(* CODESYS project arrayVar_RECOVERED_2024-06-20T13-42-02.project

Project tree, tasks and I/O mapping:
  Device : CODESYS Control Win V3, CODESYS, version 3.5.20.0
    application Application
      libraries: Standard, 3.5.18.0 (System)
      task MainTask (cyclic, interval t#20ms, priority 1) calls PLC_PRG
      function block Flash [LD]
      program PLC_PRG [ST]
*)

// Device/Application/PLC_PRG
PROGRAM PLC_PRG
VAR
	
	// This is an array which keeps the info regarding some sensors
	FArray: ARRAY[0..4] OF Bool := [TRUE, 3(FALSE), TRUE];
	// Real values from sensors
	F2: ARRAY[0..1, 0..1] OF REAL := [11, 0, 6.8, 2.3];
	F3: ARRAY[2..3, 0..1, 1..3, 0..1];
END_VAR

END_PROGRAM

// Device/Application/Flash
FUNCTION_BLOCK Flash
VAR_INPUT
	StartFlsh: BOOL;
	
END_VAR
VAR_OUTPUT
	FlashOut: BOOL;
	
	
END_VAR
VAR
	
	TON_1: TON;
	TON_0: TON;
END_VAR

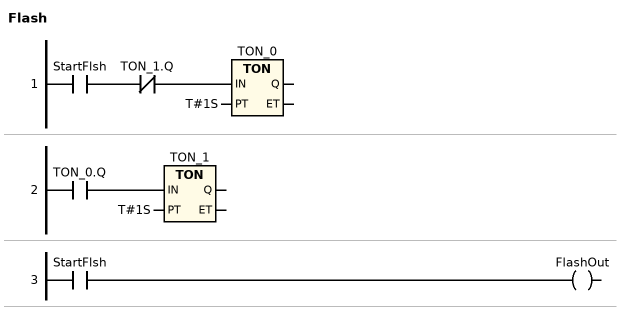
// NETWORK 1
TON_0(IN := StartFlsh AND NOT TON_1.Q, PT := T#1S); // TON

// NETWORK 2
TON_1(IN := TON_0.Q, PT := T#1S); // TON

// NETWORK 3
FlashOut := StartFlsh;

END_FUNCTION_BLOCK
